FUNCTION SetupHardware : BOOL
VAR
	iWoodBunkSlot : WoodBunk;
	iChipboardSlot : Chipboard;
	
	slotsArr : ARRAY[1..GVL.maxQueue] OF STRING;
	
	i : INT;
	j : INT;
	
	temp : INT;
END_VAR

MEMSET(ADR(slotsArr), 0, SIZEOF(slotsArr));
FOR iWoodBunkSlot:=1 TO WoodBunk.size-1 BY 1 DO //init wood bunk magazine slots
	slotsArr[iWoodBunkSlot] := TO_STRING(iWoodBunkSlot);
END_FOR
magazineLeft.setupSlots(slotsArr);
magazineRight.setupSlots(slotsArr);


MEMSET(ADR(slotsArr), 0, SIZEOF(slotsArr));
FOR iChipboardSlot:=1 TO Chipboard.size-1 BY 1 DO //init chipboard skid slots
	slotsArr[iChipboardSlot] := TO_STRING(iChipboardSlot);
END_FOR
skidLeft.setupSlots(slotsArr);
skidRight.setupSlots(slotsArr);


FOR i:=1 TO GVL.maxQueue BY 1 DO //get wood bunk magazine availability from robot
	magazineLeft.setOccupancy(i := i, occupancy := IntegerBitAccess( TO_ULINT(robotLeft.inputs[3]), TO_ULINT(i-1)) );
	skidLeft.setOccupancy(i := i, occupancy := IntegerBitAccess( TO_ULINT(robotLeft.inputs[4]), TO_ULINT(i-1)) );
	
	magazineRight.setOccupancy(i := i, occupancy := IntegerBitAccess( TO_ULINT(robotRight.inputs[3]), TO_ULINT(i-1)) );
	skidRight.setOccupancy(i := i, occupancy := IntegerBitAccess( TO_ULINT(robotRight.inputs[4]), TO_ULINT(i-1)) );
END_FOR

//enable all drives
verticalDriveLeft.bEnable := 
verticalDriveRight.bEnable := 
horizontalDriveLeft.bEnable := 
horizontalDriveRight.bEnable := 
pistonBottom.bEnable := 
TRUE;

END_FUNCTION

(* stored: Version 1.1.0.1, ProductVersion 3.1.4024.11
   POU SetupHardware: Id {ad70243f-26d6-4655-b24b-2a994d19bc18}, SpecialFunc None *)
